(* IEC 61131-3 sources: Mizera_Tube/Plc (part 15) *)

(* ---- StatMReg.plc ---- *)
#funcdec "DynMng.plc"

VAR
JUMP_INT:       LINEAR_CALC;
END_VAR

VAR_IN_OUT
PercentOutRng  AT %LSRCostK17;
END_VAR

FUNCTION_BLOCK REG_STATE_MACHINE

VAR
command:                DWORD;
State:                  DWORD;
LastCutDistance:        DWORD;
SetPointOutRange:       DWORD;      * PLC monitoring about set point out of range
RegFrozen:               BOOL;      * Regulation has been frozen from post processor
autoRegJump:             BOOL;
JumpinMode:              BOOL;
JumpinL3Mode:            BOOL;

autoRegL10:              BOOL;
L10Mode:                 BOOL;

QJump:                  DWORD;
VettYTot:               DWORD;
VettXTot:               DWORD;
VettCTot:               DWORD;

DistTot:                DWORD;
ActualDistTot:          DWORD;
ActualYDist:            DWORD;
ActualXDist:            DWORD;
ActualCDist:            DWORD;
DeltaSetPoint:          DWORD;
ZLinInterp:             DWORD;

TON_TIME_OUT:             TON;
TON_ProbeTo:              TON;
APPOGGIO:               DWORD;
appoggio:               DWORD;

firScan:                DWORD;
firScan1:               DWORD;
delScan:                DWORD;
error1:                 DWORD;
error2:                 DWORD;
error3:                 DWORD;
ToolFlt_Q_FILTERED:     DWORD;
ToolFlt_Q_FILTERED1:    DWORD;
ToolFlt_Q_FILTERED_DEL: DWORD;
ThrForOutRange:         DWORD;
SetP_S_BeforeHold:      DWORD;
tem_PercentOutRng:      DWORD;

ActualXDist_A:          DWORD;
ActualYDist_A:          DWORD;
ActualZDist_A:          DWORD;
ActualCDist_A:          DWORD;
Actual_Dist_A:          DWORD;
ActualXDist_B:          DWORD;
ActualYDist_B:          DWORD;
ActualZDist_B:          DWORD;
ActualCDist_B:          DWORD;
Actual_Dist_B:          DWORD;
Par:                   DWORD;

END_VAR

VAR_INPUT

xFirstPlcHandling:       BOOL;
xStartEx:                BOOL;
xFreezeRegol:            BOOL;         * External command to freeze regulation
xMove_Z:                   BOOL;
xHold:                   BOOL;
xFirstFirCost:          DWORD;         * ms
xSecondFirCost:         DWORD;         * ms
xDelayCost:             DWORD;         * ms
xMove_Z_SetP:             DWORD;

xProbThres:             DWORD;
xZ_TCP:                 DWORD;
xSetpoint:              DWORD;
xIsoPhase:              DWORD;         * 1: probing phase, 2: Piercing ,4: Cutting
xSensorRange:           DWORD;         * Max ange of the sensor

xNextPos_X_Jump:        DWORD;         * X setpoint coordinate for jump
xNextPos_Y_Jump:        DWORD;         * Y setpoint coordinate for jump
xNextPos_C_Jump:        DWORD;         * C setpoint coordinate for jump
xNextPos_Z_Jump:        DWORD;         * C setpoint coordinate for jump
xInit_X_Posit:          DWORD;         * X init jump position
xInit_Y_Posit:          DWORD;         * Y init jump position
xInit_C_Posit:          DWORD;         * C init jump position
xInit_Z_Posit:          DWORD;         * Z init jump position
xActual_X_Posit:        DWORD;         * X Actual position
xActual_Y_Posit:        DWORD;         * Y Actual position
xActual_C_Posit:        DWORD;         * C Actual position
xActual_Z_Posit:        DWORD;         * Z Actual position
xNextSetp:              DWORD;         * Setpoint after jump
xPrevSetp:              DWORD;         * setpoint before jump
xDistEnabRegul:         DWORD;         * Distance from target to enab regulation during jump
xZDistStopProbeJ:       DWORD;         * Z dstance to disable Probe mode during jump
xJumpReq:               BOOL;          * Jump request from ISO
xJumpL3Req:             BOOL;          * Jump L3 request from ISO
xL10Req:                BOOL;          * L10 Request from ISO
xCosBevelAngle:         DWORD;

* Surface VRTC
xSurfSignalLock:         BOOL;
xSurfaceBusy:            BOOL;
xISO_S_SimEnab:          BOOL;
xISO_S_ErrAmp:           BOOL;

* Tool VRTC

xToolSignalLock:         BOOL;
xToolBusy:               BOOL;
xISO_T_SimEnab:          BOOL;
xISO_T_ErrAmp:           BOOL;
xISO_T_SetPoint:        DWORD;
xToolFlt_Q:             DWORD;
END_VAR

VAR_OUTPUT
* Surface_VRTC_Out
y_S_SimEnab:            BOOL;             * Put Surface vrtc in Simulation
y_S_ErrAmp:             BOOL;             * Surface Error Amplifier
y_S_SetPoint:          DWORD;             * surface setpoint

* Tool_VRTC_Out
y_T_SimEnab:            BOOL;             * disable T vrtc simulation
y_T_ErrAmp:             BOOL;             * Tool Error Amplifier
y_T_SetPoint:          DWORD;

* General
yComRunning:            BOOL;
yWait:                  BOOL;
yIncSetPReached:        BOOL;
yL3SetpointReached:     BOOL;

yVPBSelect:            DWORD;
yStateMachinePhase:    DWORD;
yState:                DWORD;

END_VAR

* Reset variables at the first plc handling command

LD   xFirstPlcHandling
JMPCN no_default

LD   xFirstFirCost
DIV  %plc0.PlcCycle         * plc scan
ST   firScan

LD   xSecondFirCost
DIV  %plc0.PlcCycle         * plc scan
ST   firScan1                      **

LD   xDelayCost
DIV  %plc0.PlcCycle         * plc scan
ST   delScan                      **

LD   0
FIR_INIT (INS=1, LEN=firScan)
ST   error1

LD   0
FIR_INIT (INS=2, LEN=firScan1)
ST   error2

LD   0
DELAY_INIT (INS=1, LEN=delScan)
ST   error3
*

LD   xISO_S_SimEnab
ST   y_S_SimEnab

LD   xISO_S_ErrAmp
ST   y_S_ErrAmp

LD   xISO_T_SimEnab
ST   y_T_SimEnab

LD   xISO_T_ErrAmp
ST   y_T_ErrAmp

LD   xISO_T_SetPoint
ST   y_T_SetPoint
ST   LastCutDistance

LD   0
ST   State
ST   y_S_SetPoint                 * surface setpoint
ST   yVPBSelect
ST   yComRunning
ST   xStartEx
ST   yStateMachinePhase
ST   xJumpReq
ST   RegFrozen
ST   QJump
ST   %M180
ST   JumpinMode
ST   JumpinL3Mode
ST   yWait
ST   yIncSetPReached
ST   %PLCmsg0.8
no_default:

* Machine filters and delay model ALWAYS REFRESHED

LD   0                       * N/C
FIR_RUN (INS=1, X=xToolFlt_Q)
ST      ToolFlt_Q_FILTERED1

LD   0                       * N/C
FIR_RUN (INS=2, X=ToolFlt_Q_FILTERED1)
ST      ToolFlt_Q_FILTERED

LD   0
DELAY_RUN (INS=1,X=ToolFlt_Q_FILTERED)
DIV  10
ST  ToolFlt_Q_FILTERED_DEL

*

* Cut Distance Out of range monitoring

LD   PercentOutRng
ST   tem_PercentOutRng

LD   PercentOutRng
GT   70
OR(
LD   PercentOutRng
LT   15
)
JMPCN _SAFERNG
     LD   70
     ST   tem_PercentOutRng
_SAFERNG:

LD   xSensorRange
MULDIV (M=tem_PercentOutRng,D=1000)           * 70% del range del sensore
ST   ThrForOutRange

LD   xSetpoint
GT   ThrForOutRange
ST   SetPointOutRange

*-----------------------------------------------------------------------------------------
* Probing state machine

LD   State
EQ   0
JMPCN STATE0_end
STATE0:

 * Operative mode change

 LD    xIsoPhase
 EQ    2
 ANDN  JumpinMode
 ANDN  JumpinL3Mode
 JMPCN no_piercing_state
  LD   200                 * Piercing in progress
  ST   State
  JMP state_machine_end
 no_piercing_state:

 LD    xIsoPhase
 EQ    4
 ANDN  JumpinMode
 ANDN  JumpinL3Mode
 JMPCN no_cut_state
  LD   300                 * Cutting in progress
  ST   State
  JMP state_machine_end
 no_cut_state:

 LD    xHold
 JMPCN no_hold_sim
  LD   20                 * Go in hold condition and stop the VRTC
  ST   State
  JMP state_machine_end
 no_hold_sim:

 *
 LD    xIsoPhase
 ST    yStateMachinePhase

 *
 */////////////////////////////////////////////////////////////////////////////////
 *// Probing: vrtc wait the Z axis position threshold and disable the surface
 *// vrtc simulation and put the correct setpoint
 */////////////////////////////////////////////////////////////////////////////////

 LD    xIsoPhase
 EQ    1                                   *
 ANDN  (
 LD    xZ_TCP
 LT    xProbThres
 OR    %C18.17                             * Capacitive test in progress
 )
 AND   xStartEx
 ST    appoggio
 CAL   TON_ProbeTo(IN=appoggio,PT=10000)   * 10s
 LD    TON_ProbeTo.Q
 S     %PLCmsg0.8

 LD    xIsoPhase
 EQ    1                                   *
 AND   (
 LD    xZ_TCP
 LT    xProbThres
 OR    %C18.17                             * Capacitive test in progress
 )
 AND   xStartEx
 JMPCN STATE0_endif_A

  LD   1
  R    y_S_SimEnab                         * Put Surface vrtc in Simulation

  LD   2
  ST   yVPBSelect

  LD   xToolFlt_Q
  DIV  10
  MULDIV(M=xCosBevelAngle,D=1000)
  ST   y_S_SetPoint                        * surface setpoint

  LD   1
  ST   yComRunning

  LD  10
  ST  State
  JMP state_machine_end
 STATE0_endif_A:
*///////////////////////////////////////////////////////////////////////////////
JMP state_machine_end
STATE0_end:

LD   State
EQ   10
JMPCN STATE10_end
STATE10:
*/////////////////////////////////////////////////////////////////////////////////
*// Wait the position is reached from surface vrtc
*/////////////////////////////////////////////////////////////////////////////////

 LD    xHold
 JMPCN no_hold_real
  LD   30                 * Go in hold condition and stop the VRTC
  ST   State
  JMP state_machine_end
 no_hold_real:

 LD   xSurfSignalLock
 ANDN xSurfaceBusy
 ANDN xStartEx
 JMPCN STATE10_endif_A

  LD   0
  ST   yComRunning

  LD   0
  ST   State
  JMP state_machine_end
 STATE10_endif_A:
*///////////////////////////////////////////////////////////////////////////////
JMP state_machine_end
STATE10_end:

* During hold not allow VRTC movement

LD   State
EQ   20
JMPCN STATE20_end
STATE20:
*/////////////////////////////////////////////////////////////////////////////////
*// Hold the Z axis during the simulated descendent trajectory
*/////////////////////////////////////////////////////////////////////////////////

 LD   1
 R    y_S_ErrAmp

 LDN   xHold
 JMPCN STATE20_endif_A

  LD   1
  S    y_S_ErrAmp

  LD   0
  ST   State

  JMP state_machine_end
 STATE20_endif_A:

*///////////////////////////////////////////////////////////////////////////////
JMP state_machine_end
STATE20_end:

*
LD   State
EQ   30
JMPCN STATE30_end
STATE30:
*/////////////////////////////////////////////////////////////////////////////////
*// Hold the Z axis during the real descendent trajectory
*/////////////////////////////////////////////////////////////////////////////////

 LD   1
 R    y_S_ErrAmp

 LDN   xHold
 JMPCN STATE30_endif_A

  LD   1
  S    y_S_ErrAmp

  LD   10
  ST   State

  JMP state_machine_end
 STATE30_endif_A:

*///////////////////////////////////////////////////////////////////////////////
JMP state_machine_end
STATE30_end:

*-----------------------------------------------------------------------------------------

*-----------------------------------------------------------------------------------------
* Piercing state

LD   State
EQ   200
JMPCN STATE200_end
STATE200:
*/////////////////////////////////////////////////////////////////////////////////
*// Set piercing vpb selector
*/////////////////////////////////////////////////////////////////////////////////

 LD   xIsoPhase
 EQ   2
 ANDN xToolBusy            * update
 ANDN xSurfaceBusy         * update
 JMPCN STATE200_endif_A

  LD   3
  ST   yVPBSelect

  LD   1
 * R    y_T_SimEnab                         * Enable Tool Vrtc simulation
  S    y_T_SimEnab                         * Enable Tool Vrtc simulation

  LD   1
* S    y_S_SimEnab                         * Enable Surface vrtc Simulation
  R    y_S_SimEnab                         * Enable Surface vrtc Simulation

  LD  210
  ST  State
  JMP state_machine_end
 STATE200_endif_A:
*///////////////////////////////////////////////////////////////////////////////
JMP state_machine_end
STATE200_end:

LD   State
EQ   210
JMPCN STATE210_end
STATE210:

 * Operative mode change

 LD    xIsoPhase
 EQ    4
 JMPCN no_cut_state1
  LD    300                 * Cutting in progress
  ST    State
  JMP state_machine_end
 no_cut_state1:
*/////////////////////////////////////////////////////////////////////////////////
*// Change setpoint during piercing and synchronize the Piercing state with
*// Iso.
*/////////////////////////////////////////////////////////////////////////////////

 LD   xIsoPhase
 ST   yStateMachinePhase

 LD   xIsoPhase
 EQ   2
 AND  xStartEx
 ANDN xToolBusy
 ANDN xSurfaceBusy
 JMPCN STATE210_endif_A

  ** TEST  : in case there is a switch from out of range to in range
   LD   3
   ST   yVPBSelect
  **
  LD   1
** R    y_T_SimEnab                        * Enable Tool Vrtc simulation
  S    y_T_SimEnab                        * Enable Tool Vrtc simulation

  LD   1
** S    y_S_SimEnab                         * Enable Surface vrtc Simulation
  R    y_S_SimEnab                         * Enable Surface vrtc Simulation

  LD  SetPointOutRange                    *
  JMPCN no_sim_tool
  ** TEST
   LD   6
   ST   yVPBSelect
  **

   LD   1
   S    y_T_SimEnab                       * Enable Tool Vrtc simulation

   LD   1
*  S    y_S_SimEnab                         * Enable Surface vrtc Simulation
   S    y_S_SimEnab                         * Enable Surface vrtc Simulation

  no_sim_tool:

  LD  xSetpoint
  ST  y_T_SetPoint                        * Tool setpoint
  ST  LastCutDistance

  LD  1
  ST  yComRunning

  LD  220
  ST  State
  JMP state_machine_end
 STATE210_endif_A:
*///////////////////////////////////////////////////////////////////////////////
JMP state_machine_end
STATE210_end:

LD   State
EQ   220
JMPCN STATE220_end
STATE220:
*/////////////////////////////////////////////////////////////////////////////////
*// Setpoint reached:end of the command is set and fo to state 210 ready for
*// for next change
*/////////////////////////////////////////////////////////////////////////////////

 LD   ToolFlt_Q_FILTERED_DEL
 LT   ThrForOutRange
 AND (
  LD  LastCutDistance
  LT  ThrForOutRange
  )
 JMPCN no_setp_copy5

  LD   3
  ST   yVPBSelect

  LD   1
  R    y_S_SimEnab                         * Put Surface vrtc in Simulation

  LD   ToolFlt_Q_FILTERED_DEL
  MULDIV(M=xCosBevelAngle,D=1000)
  ST   y_S_SetPoint                       * Surface setpoint

 no_setp_copy5:

** LD   xToolSignalLock
** ANDN xToolBusy
 LD   xSurfSignalLock
 ANDN xSurfaceBusy
 ANDN xStartEx
 JMPCN STATE220_endif_A

**  LD  xSetpoint
**  ST  LastCutDistance

  LD  0
  ST  yComRunning

 ** LD   1
 ** S    y_T_SimEnab                       * Enable Tool Vrtc simulation

  LD  210
  ST  State
  JMP state_machine_end
 STATE220_endif_A:
*///////////////////////////////////////////////////////////////////////////////
JMP state_machine_end
STATE220_end:

*-----------------------------------------------------------------------------------------
* Cutting phase

LD   State
EQ   300
JMPCN STATE300_end
STATE300:

 LD  xIsoPhase
 ST  yStateMachinePhase
*/////////////////////////////////////////////////////////////////////////////////
*// This is a transition state in order to set the surface vrtc ready for
*// regulation. If the setpoint is out of range S vrtc will be in simulation.
*//
*/////////////////////////////////////////////////////////////////////////////////
 LD  xIsoPhase
 EQ  4
 ANDN xToolBusy            * update
 ANDN xSurfaceBusy         * update
 JMPCN STATE300_endif_A

  LD   1
  S    y_T_SimEnab                        * Enable Tool Vrtc simulation

  LD   1
  R    y_S_SimEnab                        * Put Surface vrtc in Simulation

  LD   4
  ST   yVPBSelect

  LD   310
  ST   State

  LD  SetPointOutRange
  JMPCN no_sim_surf
   LD   1
   S    y_S_SimEnab                       * Put Surface vrtc in Simulation
   JMP state_machine_end
  no_sim_surf:
* If the surface vrtc is in simulation not change the setpoint, otherwise it will wrong the surface position

  LD   ToolFlt_Q_FILTERED_DEL
  MULDIV(M=xCosBevelAngle,D=1000)
  ST   y_S_SetPoint                       * Surface setpoint

  JMP state_machine_end
 STATE300_endif_A:
*///////////////////////////////////////////////////////////////////////////////
JMP state_machine_end
STATE300_end:

LD   State
EQ   310
JMPCN STATE310_end
STATE310:
*/////////////////////////////////////////////////////////////////////////////////
*// Cutting mode idle: from this state is possible freeze and unfreeze regulation,
*// manage runtime setpoint change and jump request
*/////////////////////////////////////////////////////////////////////////////////

 LD   ToolFlt_Q_FILTERED_DEL
 LT   ThrForOutRange
 AND (
  LD  LastCutDistance
  LT  ThrForOutRange
  )
 ANDN RegFrozen
 ANDN L10Mode
 ANDN JumpinMode
 ANDN JumpinL3Mode
 JMPCN no_setp_copy

  LD   4
  ST   yVPBSelect

  LD   1
  R    y_S_SimEnab                         * Put Surface vrtc in Simulation

  LD   ToolFlt_Q_FILTERED_DEL
  MULDIV(M=xCosBevelAngle,D=1000)
  ST   y_S_SetPoint                       * Surface setpoint

 no_setp_copy:

* Reset L5 Routine

 LDN  xJumpReq
 JMPCN no_res_jump
  LD  1
  R   JumpinMode
 no_res_jump:

 * Reset L3 Routine

 LDN  xJumpL3Req
 JMPCN no_res_jumpL3
  LD  1
  R   JumpinL3Mode
 no_res_jumpL3:

* Reset L10 Routine

 LDN  xL10Req
 JMPCN no_res_L10
  LD  1
  R   L10Mode
 no_res_L10:

* Change operative mode to Piercing

 LD    xIsoPhase
 EQ    2
 ANDN  JumpinMode
 ANDN  JumpinL3Mode
 ANDN  L10Mode
 JMPCN no_piercing_state1
  LD   200                 * Piercing in progress
  ST   State
  JMP state_machine_end
 no_piercing_state1:

* Managment of freeze regulation from post processor
* Freeze Regulation
 LD   xFreezeRegol
 ANDN RegFrozen
 JMPCN no_freeze_en
  LD  330
  ST  State
  JMP state_machine_end *
 no_freeze_en:

* Jumping Request

 LD   xJumpReq
 ANDN JumpinMode
 ANDN JumpinL3Mode
 ANDN L10Mode
 JMPCN no_jump_req

  LD  1
  S   JumpinMode

  LD  350
  ST  State
  JMP state_machine_end
 no_jump_req:
*

* Jumping L3 Request

 LD   xJumpL3Req
 ANDN JumpinMode
 ANDN L10Mode
 JMPCN no_jump_reqL3

  LD  1
  S   JumpinL3Mode

  LD  430
  ST  State
  JMP state_machine_end
 no_jump_reqL3:
*

* L10 Request (used for cutting to piercing height)

 LD   xL10Req
 ANDN JumpinMode
 ANDN JumpinL3Mode
 ANDN L10Mode
 JMPCN no_L10_req

  LD  1
  S   L10Mode

  LD  370
  ST  State
  JMP state_machine_end
 no_L10_req:
*
* Hold Request During cut

 LD   xMove_Z
 JMPCN no_hold_req

  LD  y_S_SetPoint
  ST  SetP_S_BeforeHold

  LD  400
  ST  State
  JMP state_machine_end
 no_hold_req:

*
*/////////////////////////////////////////////////////////////////////////////////
*// If the cut distance need to be changed, this state
*// enable the simulation on the surface vrtc, disable simulation on tool vrtc
*// and set the new setpoint
*/////////////////////////////////////////////////////////////////////////////////

 LD   LastCutDistance
 NE   xSetpoint
 JMPCN STATE310_endif_A

  LD   1
  R    y_S_SimEnab                         * Put Surface vrtc in Simulation

  LD   1
  S    y_T_SimEnab                         * Enable Tool Vrtc simulation

  LD   xSetpoint
  ST   y_T_SetPoint                        * Tool setpoint
  ST   LastCutDistance                     * new

  LD   320
  ST   State

  LD  ToolFlt_Q_FILTERED_DEL
  GT  ThrForOutRange                    *
  OR  RegFrozen
  OR (
  LD  xSetpoint
  GT  ThrForOutRange
  )
  JMPCN no_sim_tool1
   ** TEST :set simulated vrtc parameters
   LD   6
   ST   yVPBSelect
   **

   LD   1
   S    y_S_SimEnab                        * Put Surface vrtc in Simulation
  JMP state_machine_end
  no_sim_tool1:

  LD   ToolFlt_Q_FILTERED_DEL
  MULDIV(M=xCosBevelAngle,D=1000)
  ST   y_S_SetPoint                       * Surface setpoint

  JMP state_machine_end
 STATE310_endif_A:

* Enable regulation Request
* This request must be here in order to not exchange the order of
* the command with the set point change

 LDN  xFreezeRegol
 AND  RegFrozen
 JMPCN no_freeze_dis
  LD  340
  ST  State
  JMP state_machine_end
 no_freeze_dis:

*///////////////////////////////////////////////////////////////////////////////
JMP state_machine_end
STATE310_end:

LD   State
EQ   320
JMPCN STATE320_end
STATE320:
*/////////////////////////////////////////////////////////////////////////////////
*// Wait the position is reached RUN-TIME. Added a  time-out condition
*/ to avoid the regulation stack on the reaching of one setpoint
*/////////////////////////////////////////////////////////////////////////////////

  LD   ToolFlt_Q_FILTERED_DEL
  LT   ThrForOutRange
  AND (
   LD  LastCutDistance
   LT  ThrForOutRange
   )
  ANDN RegFrozen
  JMPCN no_setp_copy1
   ** TEST
   LD   4
   ST   yVPBSelect
   **

   LD   1
   R    y_S_SimEnab                         * Put Surface vrtc in Simulation

   LD   ToolFlt_Q_FILTERED_DEL
   MULDIV(M=xCosBevelAngle,D=1000)
   ST   y_S_SetPoint                       * Surface setpoint
  no_setp_copy1:

  LDN  xToolSignalLock
  ANDN xToolBusy
  ST   appoggio

* Time-out is mandatory, in order to avoid the regulation keep this state
* and saturate the vrtc limit

  CAL  TON_TIME_OUT (IN:=appoggio,PT:=250)

  LD   xToolSignalLock
  ANDN xToolBusy
  OR   TON_TIME_OUT.Q
  JMPCN STATE320_endif_A
    ** TEST
    LD   4
    ST   yVPBSelect
    **

    LD   1
    R    y_S_SimEnab                         * Put Surface vrtc in Simulation

    LD   1
    S    y_T_SimEnab                         * Enable Tool Vrtc simulation

    LD   310
    ST   State

    LD  SetPointOutRange               **** Verificare se va aggiornato con le condizioni fatte per gli altri stati
    OR  RegFrozen
    JMPCN no_sim_surf1
     ** TEST
     LD   6
     ST   yVPBSelect
     **

     LD   1
     S    y_S_SimEnab                       * Put Surface vrtc in Simulation
     JMP state_machine_end
    no_sim_surf1:

* If the surface vrtc is in simulation not change the setpoint, otherwise it will wrong the surface position

   LD   ToolFlt_Q_FILTERED_DEL
   MULDIV(M=xCosBevelAngle,D=1000)
   ST   y_S_SetPoint                       * Surface setpoint

 JMP state_machine_end
 STATE320_endif_A:
*///////////////////////////////////////////////////////////////////////////////
JMP state_machine_end
STATE320_end:

LD   State
EQ   330
JMPCN STATE330_end
STATE330:
*/////////////////////////////////////////////////////////////////////////////////
*// Enable the simulation of the sensor when post processor need freeze
*// the height control
*/////////////////////////////////////////////////////////////////////////////////

 ** TEST
 LD   6
 ST   yVPBSelect
 **

 LD  1
 S   y_S_SimEnab                       * Put Surface vrtc in Simulation

 LD  1
 S   y_T_SimEnab                         * Enable Tool Vrtc simulation

 LD  1
 S   RegFrozen

 LD  310
 ST  State

 JMP state_machine_end
STATE330_endif_A:
*///////////////////////////////////////////////////////////////////////////////
JMP state_machine_end
STATE330_end:

LD   State
EQ   340
JMPCN STATE340_end
STATE340:
*/////////////////////////////////////////////////////////////////////////////////
*// Post processor command regulation again, but need to be careful about set point
*// if it is inside the range, surface can back to regulate otherwise no
*/////////////////////////////////////////////////////////////////////////////////

  LD   ToolFlt_Q_FILTERED_DEL
  LT   ThrForOutRange
  AND (
   LD  LastCutDistance
   LT  ThrForOutRange
   )
 JMPCN no_remove_sim_S
  ** TEST
  LD   4
  ST   yVPBSelect
  **

  LD  1
  R   y_S_SimEnab                        * Surface vrtc in Simulation

* Need give setpoint because if it change distance when is frozen and setpoint is inside the range
* it is not refresced on surface regulator

  LD   ToolFlt_Q_FILTERED_DEL
  MULDIV(M=xCosBevelAngle,D=1000)
  ST   y_S_SetPoint                      * Surface setpoint

 no_remove_sim_S:

 LD  1
 S   y_T_SimEnab                         * Enable Tool Vrtc simulation

 LD  1
 R   RegFrozen

 LD  310
 ST  State

 JMP state_machine_end
STATE340_endif_A:
*///////////////////////////////////////////////////////////////////////////////
JMP state_machine_end
STATE340_end:

* Jump
LD   State
EQ   350
JMPCN STATE350_end
STATE350:
*/////////////////////////////////////////////////////////////////////////////////
*// Jump Request: select VPBselect at 1 for jump column,put vrtc surface in
*// simulation. The algorithm calulates the setpoint for Surface and Tool
*// Vrtc. Surface will perform the parabolic trajectory, the Tool will apply the
*// setpoint change
*/////////////////////////////////////////////////////////////////////////////////
 LD  xStartEx
 JMPCN no_start_jump

  LD   1
  ST   yComRunning

  LD   1
  ST   yVPBSelect

  LD   1
  S    y_S_SimEnab              * Surface vrtc in Simulation

  LD   xNextPos_Y_Jump         * Y setpoint coordinate for jump
  SUB  xInit_Y_Posit           * Y init jump position
  ABS
  ST   VettYTot                * Distance in Y direction

  LD   xNextPos_X_Jump         * X setpoint coordinate for jump
  SUB  xInit_X_Posit           * X init jump position
  ABS
  ST   VettXTot                * Distance in X direction

  LD   0
  ST   VettCTot                      ** Distance in C direction

  LD   xNextPos_C_Jump
  SUB  xInit_C_Posit
  ABS
  ST   VettCTot                      ** Distance in C direction

  LD   0
  HYPOT (X=VettXTot,Y=VettYTot)
  ST   DistTot                 * total distance for jump

  LD   0
  HYPOT (X=DistTot,Y=VettCTot)       ** total distance for jump
  ST   DistTot                       ** total distance for jump

  LD   xActual_X_Posit
  SUB  xInit_X_Posit                 * X init jump position
  ABS
  ST   ActualXDist

  LD   xActual_Y_Posit               * Y Actual position
  SUB  xInit_Y_Posit                 * Y init jump position
  ABS
  ST   ActualYDist

  LD   xActual_C_Posit
  SUB  xInit_C_Posit
  ABS
  ST   ActualCDist

  LD   0
  HYPOT (X=ActualXDist,Y=ActualYDist)
  ST   ActualDistTot

  LD   0
  HYPOT (X=ActualDistTot,Y=ActualCDist)
  ST   ActualDistTot
  ST   %M181

  * Calcolo quota per jumping mode

  LD   ActualDistTot
  ST   JUMP_INT.xInput               * Distance to go

  LD   130
  ST   JUMP_INT.xIndex               * cut line index (initial value 1 to 10)

  CAL  JUMP_INT

  LD   JUMP_INT.yResult              * Result
  DIV  10
  ST   QJump                         ** Quota Z per Jumping

  LD   xPrevSetp                      * setpoint before jump
  DIV  10
  ADD  QJump
  ST   y_S_SetPoint
  ST   %M184

  ************************************************************************************
*  Algorithm for auto jump regulation enable
*  and setpoint changing compensation

  LD   xNextSetp                * Setpoint after jump
  SUB  xPrevSetp                * setpoint before jump
  ST   DeltaSetPoint

* TEST
 * LD   ActualDistTot
 * MUL  2
 * ST   APPOGGIO

 * LD   APPOGGIO
 * GT   DistTot
 * JMPCN forcedist
 *  LD   DistTot
 *  ST   APPOGGIO
 * forcedist:
***
 * LD   APPOGGIO
  LD   ActualDistTot
  MULDIV (M=DeltaSetPoint,D=DistTot) ** total distance for jump
  DIV  10                            *cmm
  ST   ZLinInterp

  LD   xPrevSetp                * setpoint before jump
  DIV  10
  ADD  ZLinInterp
  ST   y_T_SetPoint

  ** Test of regulation on fly

  LD   DistTot                       ** total distance for jump
  SUB  ActualDistTot                 * Actual total distance by measured speed
  LE   xDistEnabRegul                * Distance from target to enab regulation
  ST   autoRegJump                   ** During jump allow auto regulation on

  LD   autoRegJump
  JMPCN no_jump_end

    LD  xZ_TCP
    GT  xZDistStopProbeJ             * distance along Z to disable the probe vpbselector during jump
    JMPCN no_Zover_range

     LD  0
     ST  yVPBSelect

     LD   xPrevSetp                * setpoint before jump
     DIV  10
     MULDIV(M=xCosBevelAngle,D=1000)
     ST  y_S_SetPoint

    JMP no_jump_end
    no_Zover_range:

    LD  1
    R   y_S_SimEnab                 * Surface vrtc in Simulation

    LD  2
    ST  yVPBSelect

    LD   ToolFlt_Q_FILTERED_DEL
    MULDIV(M=xCosBevelAngle,D=1000)
    ST  y_S_SetPoint
    ST  %M183

  no_jump_end:
 no_start_jump:

 LDN  xJumpReq
 JMPCN no_end_jump

  LD  1
  R   y_S_SimEnab                 * Surface vrtc in Simulation

  LD  2
  ST  yVPBSelect

  LD   ToolFlt_Q_FILTERED_DEL
  MULDIV(M=xCosBevelAngle,D=1000)
  ST  y_S_SetPoint

  LD  360
  ST  State
 no_end_jump:

 JMP state_machine_end
STATE350_endif_A:
*///////////////////////////////////////////////////////////////////////////////
JMP state_machine_end
STATE350_end:

LD   State
EQ   360
JMPCN STATE360_end
STATE360:
*/////////////////////////////////////////////////////////////////////////////////
*// Wait the position is reached after jump
*/////////////////////////////////////////////////////////////////////////////////

 LD   ToolFlt_Q_FILTERED_DEL
 MULDIV(M=xCosBevelAngle,D=1000)
 ST  y_S_SetPoint

 LD   xSurfSignalLock
 ANDN xSurfaceBusy
 ANDN xStartEx
 JMPCN STATE360_endif_A

    LD   0
    ST   yComRunning

    LD   xNextSetp                * Setpoint after jump
    DIV  10
    ST   LastCutDistance

    LD   1                        * Reset bit to enable always regulation after jump
    R    RegFrozen

    LD   310
    ST   State
 JMP state_machine_end
STATE360_endif_A:
*///////////////////////////////////////////////////////////////////////////////
JMP state_machine_end
STATE360_end:

LD   State
EQ   370
JMPCN STATE370_end
STATE370:
*/////////////////////////////////////////////////////////////////////////////////
*// This state manage the L10 cutting transition, to reach the set point it is only
*// interpolated the Tool VRTC from cutting position to Piercing position.
*/////////////////////////////////////////////////////////////////////////////////

 LD  xStartEx
 JMPCN no_start_L10

  LD   1
  ST   yComRunning

  LD   1
  ST   yVPBSelect

  LD   1
  S    y_S_SimEnab              * Surface vrtc in Simulation

  LD   xNextPos_Y_Jump         * Y setpoint coordinate for jump
  SUB  xInit_Y_Posit           * Y init jump position
  ABS
  ST   VettYTot                * Distance in Y direction

  LD   xNextPos_X_Jump         * X setpoint coordinate for jump
  SUB  xInit_X_Posit           * X init jump position
  ABS
  ST   VettXTot                * Distance in X direction

  LD   0
  HYPOT (X=VettXTot,Y=VettYTot)
  ST   DistTot                 * total distance for jump

  LD   xActual_X_Posit
  SUB  xInit_X_Posit                 * X init jump position
  ABS
  ST   ActualXDist

  LD   xActual_Y_Posit               * Y Actual position
  SUB  xInit_Y_Posit                 * Y init jump position
  ABS
  ST   ActualYDist

  LD   0
  HYPOT (X=ActualXDist,Y=ActualYDist)
  ST   ActualDistTot
  ST   %M181

  ************************************************************************************
*  Algorithm for auto jump regulation enable
*  and setpoint changing compensation

  LD   xNextSetp                * Setpoint after jump
  SUB  xPrevSetp                * setpoint before jump
  ST   DeltaSetPoint

* TEST
 * LD   ActualDistTot
 * MUL  2
 * ST   APPOGGIO

 * LD   APPOGGIO
 * GT   DistTot
 * JMPCN forcedist1
 *  LD   DistTot
 *  ST   APPOGGIO
 * forcedist1:
***
  *LD   APPOGGIO
  LD   ActualDistTot
  MULDIV (M=DeltaSetPoint,D=DistTot) ** total distance for jump
  DIV  10                            *cmm
  ST   ZLinInterp

  LD   xPrevSetp                * setpoint before jump
  DIV  10
  ADD  ZLinInterp
  ST   y_T_SetPoint

  ** Test of regulation on fly

  LD   DistTot                       ** total distance for jump
  SUB  ActualDistTot                 * Actual total distance by measured speed
  LE   xDistEnabRegul                * Distance from target to enab regulation
  ST   autoRegL10                   ** During jump allow auto regulation on

  LD   autoRegL10
  JMPCN no_L10_end

    LD  1
    R   y_S_SimEnab                 * Surface vrtc in Simulation

    LD  2
    ST  yVPBSelect

    LD   ToolFlt_Q_FILTERED_DEL
    MULDIV(M=xCosBevelAngle,D=1000)
    ST  y_S_SetPoint
    ST  %M183

  no_L10_end:
 no_start_L10:

 LDN  xL10Req
 JMPCN no_end_L10

  LD  1
  R   y_S_SimEnab                 * Surface vrtc in Simulation

  LD  2
  ST  yVPBSelect

  LD   ToolFlt_Q_FILTERED_DEL
  MULDIV(M=xCosBevelAngle,D=1000)
  ST  y_S_SetPoint

  LD  380
  ST  State
 no_end_L10:

 JMP state_machine_end
STATE370_endif_A:
*///////////////////////////////////////////////////////////////////////////////
JMP state_machine_end
STATE370_end:
*
LD   State
EQ   380
JMPCN STATE380_end
STATE380:
*/////////////////////////////////////////////////////////////////////////////////
*// Wait the position is reached after L10
*/////////////////////////////////////////////////////////////////////////////////

 LD   ToolFlt_Q_FILTERED_DEL
 MULDIV(M=xCosBevelAngle,D=1000)
 ST  y_S_SetPoint

 LD   xSurfSignalLock
 ANDN xSurfaceBusy
 ANDN xStartEx
 JMPCN STATE380_endif_A

    LD   0
    ST   yComRunning

    LD   xNextSetp                * Setpoint after jump       CAMBIARE NOME
    DIV  10
    ST   LastCutDistance

    LD   310
    ST   State
 JMP state_machine_end
STATE380_endif_A:
*///////////////////////////////////////////////////////////////////////////////
JMP state_machine_end
STATE380_end:

* Hold

LD   State
EQ   400
JMPCN STATE400_end
STATE400:
*///////////////////////////////////////////////////////////////////////////////////
*// Hold management: Z is moved according the Z inc movement; when xZmove is
*// removed, the Z back in the prevous point. If the operator move by retrace
*// the tool setpoint is updated run-time, the freeze conditition due to the
*// M82 M83 or distance out of range that can happen during the retrace are managed.
*///////////////////////////////////////////////////////////////////////////////////

  LD  1
  S   y_S_SimEnab                 * Surface vrtc in Simulation

  LD  xMove_Z_SetP
  ST  y_S_SetPoint

  LD  5
  ST  yVPBSelect

  LD  xSetpoint
  ST  y_T_SetPoint
  ST  LastCutDistance

  LD  xFreezeRegol
  ST  RegFrozen

  LDN  yIncSetPReached
  JMPCN no_wait_incSetp
    LD   410
    ST   State
    JMP  state_machine_end
  no_wait_incSetp:

  LDN  xMove_Z
  JMPCN no_return_pause

    LD  1
    S   yWait

* IF stand-off is in capacitive range

    LD  ToolFlt_Q_FILTERED_DEL
    LT  ThrForOutRange
    AND (
    LD  LastCutDistance
    LT  ThrForOutRange
    )
    ANDN RegFrozen
    JMPCN no_setp_copy3
    ** TEST
     LD   5
     ST   yVPBSelect
    **
     LD   1
     R    y_S_SimEnab                        * Put Surface vrtc in Simulation

     LD   ToolFlt_Q_FILTERED_DEL
     MULDIV(M=xCosBevelAngle,D=1000)
     ST   y_S_SetPoint                       * Surface setpoint

     LD   420
     ST   State
    JMP state_machine_end
    no_setp_copy3:

    LD  ToolFlt_Q_FILTERED_DEL
    GT  ThrForOutRange
    OR (
    LD  LastCutDistance
    GT  ThrForOutRange
    )
    OR  RegFrozen
    JMPCN no_setp_copy4

     **
     LD   5
     ST   yVPBSelect
     **
     LD   1
     S    y_S_SimEnab                        * Put Surface vrtc in Simulation

     LD   SetP_S_BeforeHold
     ST   y_S_SetPoint                       * Surface setpoint

     LD   420
     ST   State
     JMP state_machine_end
    no_setp_copy4:

  no_return_pause:

 STATE400_endif_A:
*///////////////////////////////////////////////////////////////////////////////
JMP state_machine_end
STATE400_end:

LD   State
EQ   410
JMPCN STATE410_end
STATE410:
*/////////////////////////////////////////////////////////////////////////////////
*// Wait Z reach the setpoint from inc movement
*/////////////////////////////////////////////////////////////////////////////////

 LD   xSurfSignalLock
 ANDN xSurfaceBusy
 JMPCN STATE410_endif_A

  LD   1
  S    yIncSetPReached

  LD   400
  ST   State

 STATE410_endif_A:
*///////////////////////////////////////////////////////////////////////////////
JMP state_machine_end
STATE410_end:

LD   State
EQ   420
JMPCN STATE420_end
STATE420:
*/////////////////////////////////////////////////////////////////////////////////
*// Wait the position is reached after return from hold
*/////////////////////////////////////////////////////////////////////////////////

 LD   xSurfSignalLock
 ANDN xSurfaceBusy
 JMPCN STATE420_endif_A

  LD   1
  R    yWait

  LD   1
  R    yIncSetPReached

  LD   310
  ST   State

 STATE420_endif_A:
*///////////////////////////////////////////////////////////////////////////////
JMP state_machine_end
STATE420_end:

* Jump L3 Between Sides
LD   State
EQ   430
JMPCN STATE430_end
STATE430:
*/////////////////////////////////////////////////////////////////////////////////
*// Jump L3 Request: VRTC is in simulation state, and must wait that interpolation
*// finish. Basically works like L5 but there is oly the interpolation of the
*// set-point but parabolic movement is done by the interpolator.
*/////////////////////////////////////////////////////////////////////////////////
 LD  xStartEx
 JMPCN no_start_jump1

  LD   1
  ST   yComRunning

  LD   6
  ST   yVPBSelect

  LD   1
  S    y_S_SimEnab              * Surface vrtc in Simulation

* Calculate vector A

  LD   xActual_X_Posit
  SUB  xInit_X_Posit                 * X init jump position
  DIV  100
  ABS
  ST   ActualXDist_A

  LD   xActual_Y_Posit
  SUB  xInit_Y_Posit                 * Y init jump position
  DIV  100
  ABS
  ST   ActualYDist_A

  LD   xActual_Z_Posit
  SUB  xInit_Z_Posit                 * Z init jump position
  DIV  100
  ABS
  ST   ActualZDist_A

  LD   xActual_C_Posit
  SUB  xInit_C_Posit                 * C init jump position
  DIV  100
  ABS
  ST   ActualCDist_A

* || A ||

  LD   ActualXDist_A
  MUL  ActualXDist_A
  ADD (
  LD   ActualYDist_A
  MUL  ActualYDist_A
  )
  ADD (
  LD   ActualZDist_A
  MUL  ActualZDist_A
  )
  ADD (
  LD   ActualCDist_A
  MUL  ActualCDist_A
  )
  ST   Actual_Dist_A

  LD   Actual_Dist_A
  SQRT
  ST   Actual_Dist_A

* Calculate vector B

  LD   xActual_X_Posit
  SUB  xNextPos_X_Jump                 * X Next jump position
  DIV  100
  ABS
  ST   ActualXDist_B

  LD   xActual_Y_Posit
  SUB  xNextPos_Y_Jump                 * Y Next jump position
  DIV  100
  ABS
  ST   ActualYDist_B

  LD   xActual_Z_Posit
  SUB  xNextPos_Z_Jump                 * Z Next jump position
  DIV  100
  ABS
  ST   ActualZDist_B

  LD   xActual_C_Posit
  SUB  xNextPos_C_Jump                 * C Next jump position
  DIV  100
  ABS
  ST   ActualCDist_B

* || B ||

  LD   ActualXDist_B
  MUL  ActualXDist_B
  ADD (
  LD   ActualYDist_B
  MUL  ActualYDist_B
  )
  ADD (
  LD   ActualZDist_B
  MUL  ActualZDist_B
  )
  ADD (
  LD   ActualCDist_B
  MUL  ActualCDist_B
  )
  ST   Actual_Dist_B

  LD   Actual_Dist_B
  SQRT
  ST   Actual_Dist_B

* Par = (|| A ||) / ( || A || + || B || )

  LD   Actual_Dist_A
  MUL  100
  DIV  (
  LD   Actual_Dist_A
  ADD  Actual_Dist_B
  )
  ST   Par

  LD   xPrevSetp                      * setpoint before jump
  DIV  10
  ST   y_S_SetPoint
  ST   %M184

  LD   xNextSetp                * Setpoint after jump
  SUB  xPrevSetp                * setpoint before jump
  ST   DeltaSetPoint

  *LD   ActualDistTot
  *MULDIV (M=DeltaSetPoint,D=DistTot) ** total distance for jump
  *DIV  10                            *cmm
  *ST   ZLinInterp

  LD   Par
  MULDIV (M=DeltaSetPoint,D=100) ** total distance for jump
  DIV  10                            *cmm
  ST   ZLinInterp

  LD   xPrevSetp                * setpoint before jump
  DIV  10
  ADD  ZLinInterp
  ST   y_T_SetPoint

  LD   Par
  GE   100
  *ST   %M189.1
  ST   yL3SetpointReached

 no_start_jump1:

 LDN  xJumpL3Req
 JMPCN no_end_jump1

  LD  1
  R   y_S_SimEnab                 * Surface vrtc in Simulation

  LD  3
  ST  yVPBSelect

  LD   ToolFlt_Q_FILTERED_DEL
  MULDIV(M=xCosBevelAngle,D=1000)
  ST  y_S_SetPoint

  LD  440
  ST  State
 no_end_jump1:

 JMP state_machine_end
STATE430_endif_A:
*///////////////////////////////////////////////////////////////////////////////
JMP state_machine_end
STATE430_end:

LD   State
EQ   440
JMPCN STATE440_end
STATE440:
*/////////////////////////////////////////////////////////////////////////////////
*// Wait the position is reached after jump
*/////////////////////////////////////////////////////////////////////////////////

 LD  1
 R   y_S_SimEnab                 * Surface vrtc in Simulation

 LD   ToolFlt_Q_FILTERED_DEL
 MULDIV(M=xCosBevelAngle,D=1000)
 ST  y_S_SetPoint

 LD   xSurfSignalLock
 ANDN xSurfaceBusy
 ANDN xStartEx
 JMPCN STATE440_endif_A

    LD   0
    ST   yComRunning

    LD   xNextSetp                * Setpoint after jump
    DIV  10
    ST   LastCutDistance

 *  LD   1                        * Reset bit to enable always regulation after jump
 *  R    RegFrozen

    LD   310
    ST   State
 JMP state_machine_end
STATE440_endif_A:
*///////////////////////////////////////////////////////////////////////////////
JMP state_machine_end
STATE440_end:

state_machine_end:
IDLE_end:

LD   State
ST   yState
ST   %M182

LD   y_S_SetPoint
ST   %M180

LD   y_T_SetPoint
ST   %M192

LD   LastCutDistance
ST   %M190

LD   xSetpoint
ST   %M191

END_FUNCTION_BLOCK

(* ---- SupForce.plc ---- *)
#funcdec "DynMng.plc"
#funcdec "FBAux.plc"

*//============================================================================
*// Force Following Support to be Down from ISO management
*//============================================================================

FUNCTION_BLOCK     ISO_SUP_FORCE_DOWN

VAR_INPUT
xIsoForce:         BOOL;      * iso_LsronCutting
xHoldMovSuperv:    BOOL;      * yHoldMovSuperv
END_VAR

VAR
Sup_Up_NotAllow:   BOOL;
R_TRIG_DWNCMD:     R_TRIG;
END_VAR

VAR_OUTPUT
yForceDwn:         BOOL;
END_VAR

CAL    R_TRIG_DWNCMD(CLK=xHoldMovSuperv)
LD     xIsoForce
AND    R_TRIG_DWNCMD.Q
S      Sup_Up_NotAllow

LDN    xIsoForce
ORN    %cn0.rc8.0
JMPCN  CLRSTATE
LD     %PLCFLAGS.0
ST     Sup_Up_NotAllow
CLRSTATE:

LD     Sup_Up_NotAllow
AND    xIsoForce
AND    %cn0.rc8.0
ST     yForceDwn

END_FUNCTION_BLOCK

*//============================================================================
*// In case of slave axis gearing state of G4010,
*// %ra92 == %ra24
*// PLC pre-stop quota need to be added (Estimated without JERK calculation)
*// CAL CALQ_PRESSLV(xEn:=,xQta:=,xSpdNum:=)
*// 0.5G 50000 Jerk as bench mark
*//============================================================================

FUNCTION_BLOCK     CALQ_PRESSLV

VAR_INPUT
xEn:               BOOL;
xQta:              DWORD;      * %ra4 / ra92
xSpdNum:           DWORD;      * The spline table number
END_VAR

VAR
tem_dis:           DWORD;
QtaCalc:           POINTS_INT_CALC;
END_VAR

VAR_OUTPUT
Q:                 DWORD;
END_VAR

LD     xQta
ST     Q

* Pre simpling data 0.5g 50000 Jerk，when RA92 fails

* speed > 2.2m/min and xQta < 1mm

LD     %ra115
MULDIV(M=60,D=1000)
GT     2200
AND(
       LD   xQta
       SUB  %ra24
	   LT   1000
)
JMPCN _ACT_LINERA
       LD   %ra115
       MULDIV(M=60,D=1000)
       ABS
       ST   QtaCalc.xPercSpeed            * Speed percentual value

       LD   1
       ST   QtaCalc.xCutLineInd           * cut line index (initial value 1 to 10)

       LD   xSpdNum
       ST   QtaCalc.xCodTec               * Tecnology 0=duty 1=power 2=frequency

       CAL  QtaCalc

       LD   QtaCalc.yResult               * Result
	   ST   tem_dis

	   LD   tem_dis
	   LT   0
	   JMPCN _SAFTY
	        LD  0
			ST  tem_dis
	   _SAFTY:

	   LD   tem_dis
	   ADD  xQta
       ST   Q

	   LDN  %ra3.2                        * Forward Movement of Slave Spindle
       ANDN %ra3.0
       JMPCN BCKWARDX1CASE
	        LD   xQta
            SUB  tem_dis
            ST   Q
       BCKWARDX1CASE:
_ACT_LINERA:

* Vel   Dis
* 2500	3020
* 5000	6320
* 7500	9965
* 10000	13955
* 12500	18297
* 15000	22985
* 17500	28020
* 20000	33400
* 22500	39128
* 25000	45200
* 27500	51626
* 30000	58396
* 32500	65516
* 35000	72980
* 37500	80792
* 40000	88950
* 42500	97459
* 45000	106313
* 47500	115513
* 50000	125000

PATH   %pd_splines[xSpdNum]

LD     %PLCFLAGS.8
JMPCN  _INIGLB
       LD  2
       ST  %pdh_interpType
       LD  21
       ST  %pdh_nPoints

       LD  0
       ST  %pdh_X0
       ST  %pdh_Y0

       LD  2500
       ST  %pdh_X1
	   LD  3020
       ST  %pdh_Y1

	   LD  5000
       ST  %pdh_X2
	   LD  6320
       ST  %pdh_Y2

	   LD  7500
       ST  %pdh_X3
	   LD  9965
       ST  %pdh_Y3

	   LD  10000
       ST  %pdh_X4
	   LD  13955
       ST  %pdh_Y4

	   LD  12500
       ST  %pdh_X5
	   LD  18297
       ST  %pdh_Y5

	   LD  15000
       ST  %pdh_X6
	   LD  22985
       ST  %pdh_Y6

	   LD  17500
       ST  %pdh_X7
	   LD  28020
       ST  %pdh_Y7

	   LD  20000
       ST  %pdh_X8
	   LD  33400
       ST  %pdh_Y8

	   LD  22500
       ST  %pdh_X9
	   LD  39128
       ST  %pdh_Y9

	   LD  25000
       ST  %pdh_X10
	   LD  45200
       ST  %pdh_Y10

	   LD  27500
       ST  %pdh_X11
	   LD  51626
       ST  %pdh_Y11

	   LD  30000
       ST  %pdh_X12
	   LD  58396
       ST  %pdh_Y12

	   LD  32500
       ST  %pdh_X13
	   LD  65516
       ST  %pdh_Y13

	   LD  35000
       ST  %pdh_X14
	   LD  72980
       ST  %pdh_Y14

	   LD  37500
       ST  %pdh_X15
	   LD  80792
       ST  %pdh_Y15

	   LD  40000
       ST  %pdh_X16
	   LD  88950
       ST  %pdh_Y16

	   LD  42500
       ST  %pdh_X17
	   LD  97459
       ST  %pdh_Y17

	   LD  45000
       ST  %pdh_X18
	   LD  106313
       ST  %pdh_Y18

	   LD  47500
       ST  %pdh_X19
	   LD  115513
       ST  %pdh_Y19

	   LD  50000
       ST  %pdh_X20
	   LD  125000
       ST  %pdh_Y20

_INIGLB:

END_FUNCTION_BLOCK

*//============================================================================
*// Cylinder Composite Support Calculation Based On Current Profile Shape
*// CAL CALC_CYCOMSUP(xLenCy:=, xEnCyTubeSiz:=)
*//============================================================================

FUNCTION_BLOCK     CALC_CYCOMSUP

VAR_INPUT
xLenCy:            DWORD;     * The stroke of cylinder [mm]
xEnCyTubeSiz:      DWORD;     * > Qta to disable cylinder [mm] (not the trave of servo because which could be different)
xAxNum:            DWORD;     * The servo support axis number
END_VAR

VAR
OutofRng:          BOOL;
X:                 DWORD;
Y:                 DWORD;
Radius:            DWORD;
inner:             DWORD;
outter:            DWORD;
temLenCy:          DWORD;
temAxtra:          DWORD;
CyTubeSiz:         DWORD;
MaxMin:          COMPARE;
END_VAR

VAR_OUTPUT
* Bit 0: Only Motor, offset == 0
* Bit 1: Both Cylinder and Motor, offset == Cylinder Stroke
* Bit 2: Impossible to always follow, msgout (Out of range, should not happen. Otherwise, tube is too large)
yModeCode:         DWORD;
END_VAR

LD     xLenCy
MUL    1000
ST     temLenCy

LD     xEnCyTubeSiz
MUL    1000
ST     CyTubeSiz

LD     %gIso23
MUL    1000
ST     X

LD     %gIso24
MUL    1000
ST     Y

CAL    MaxMin(A:=X,B:=Y)
LD     MaxMin.yMin
DIV    2
ST     inner

LD     0
HYPOT (X=X,Y=Y)
DIV    2
ST     outter

LD     %gIso25       *RAIDIUS UNIT DIFFERENT
ST     Radius

LD     %gIso26
EQ     0
JMPCN  _RECT
       LD  X
	   SUB Radius
	   ST  X

	   LD  Y
	   SUB Radius
	   ST  Y

       LD  0
       HYPOT(X=X,Y=Y)
	   DIV 2
       ADD Radius
	   ST  outter
_RECT:

LD     %gIso26
EQ     1
JMPCN  _ROUND
       LD  inner
	   ST  outter
_ROUND:

* Output

LD     0
ST     yModeCode

PATH   %ax[xAxNum]

LD     %pa22
SUB    %pa21
ST     temAxtra

LD     outter
SUB    inner
GT(
LD     temAxtra
SUB    temLenCy
)
AND(
LD     temLenCy
GT     inner
)
AND(
LD     temLenCy
LT     outter
)
ST     OutofRng

LD     outter
GT     CyTubeSiz
ST     yModeCode.0
STN    yModeCode.1

LD     OutofRng
ST     yModeCode.2

END_FUNCTION_BLOCK

(* ---- suppFB.plc ---- *)
*******************************************************************************
*   suppFB.plc
*   ESAutomotion
*   LASER machine
*******************************************************************************
#funcdec "assi.plc"

*******************************************************************************
*   Support axis management (Cascading Blend Switch, G.D)
*******************************************************************************

VAR_IN_OUT
AxPos             AT  %ra4;      * Axis position
Go_Follow         AT  %rgau0;    * Force down by blending algh.
AddFollow         AT  %rgau1;    * Add value during following
BldState          AT  %rgau2;    * Blend switch output, (0->1000) (parking -> following)
ParkingSet        AT  %rgau3;    * Real time parking position (input)
AddFollow_Out     AT  %rgau4;    * Add value during following (output)
ParkingSet_Out    AT  %rgau5;    * Real time parking position (output)

filterT1Rate      AT  %rgdau0;   * Blendswitch filter rate [0.001/min]
addValueVel       AT  %rgdau1;   * Following add value speed [um/min]
addValueVelM      AT  %rgdau2;   * Parking speed [um/min]

ProbeThreshold    AT  %gIso30;   *(gIso30) probe threshold (G2292)

LatCenterToCloseRun AT %SUPPORTS_SYSTEM.values13.17;
END_VAR

FUNCTION_BLOCK    SUPPORT

VAR_INPUT
xUaxDir:          BOOL;          * 1 - if spindle move towards the 0 of the machine decreasing its quota
                                 * 0 - if spindle move towards the 0 of the machine increasing its quota
xHoldExem:        BOOL;          * Support Hold Exemption (in case of initialization)
xUaxStill:        BOOL;          * U axis is not moving (%ra3.0)
xReset:           BOOL;          * Emergency and Reset for PosAx
xEnabAutoDwn:     BOOL;          * Enable Auto Support Down
xEnabAutoUp:      BOOL;          * Enable Auto Support Up (Blend)
xBlendSwitchEn:   BOOL;          * blendswitch enable
xParkCmd:         BOOL;          * JOG / Auto Cmd to park
xSensSafePos:     BOOL;          * Safety sensor to be sure the support is parked
xEnSecFollow:     BOOL;          * Enable addvalue during support following
xG520VSup:        BOOL;          * In G520 using V support unloading (Parking Target by ISO)
xEnCyComSup:      BOOL;          * Enable motor cylinder composite support
xEnBldFeed:       BOOL;          * Blend switch feedrate management

xSupervisePos:   DWORD;          * Position of the U axis -> start autodown
xSuperviseOft:   DWORD;          * Offset of position U to be closer to the support
xLimitSuppDwn:   DWORD;          * U axis limit position for support down
xParkingPos:     DWORD;          * Support Parking position
xUnSupQta:       DWORD;          * Support Parking position to Unload
xAddFollPos:     DWORD;          * Added following targets
xCyComOft:       DWORD;          * Motor cylinder composite support blend switch offset
xM700_M704:      DWORD;          * M700, M704 executing
xBlendId:        DWORD;          * Blend ID for speed reset ([lv, lat, ulv, uhor]=[0,1,2,3])
xBldFeed:        DWORD;          * Blend switch feedrate % (0-100)
END_VAR

VAR_OUTPUT
yReqGrant:        BOOL;
yHoldMovSupp:     BOOL;
yHoldMovSuperv:   BOOL;
yAxInParkPos:     BOOL;
yCenterOpen:      BOOL;
yCyComDwn:        BOOL;
yCyComOft:       DWORD;
END_VAR

VAR
resReq:           BOOL;
Req_Parking:      BOOL;
HoldSuppAxis:     BOOL;
HoldSuperviAxis:  BOOL;
appoggio:         BOOL;
GoUpSuppAuto:     BOOL;
M700Running:      BOOL;
M704Running:      BOOL;
CenterOpen:       BOOL;

OuterPlusOne:     DWORD;
Supervise_Oft:    DWORD;
ProbeThrsTmp:     DWORD;

TON_CLOSE_LOOP:    TON;
TRIG_PRKCON:      TRIG;
R_TRIG_BLD:     R_TRIG;
R_RES_REQ:      R_TRIG;
RTRIG_REQ_PARK: R_TRIG;
RTRIG_PARK:     R_TRIG;
RTRIG_RES_PARK: R_TRIG;
RTRIG_SAFE_DWN: R_TRIG;
RTRIG_REQ_UP:   R_TRIG;
RTRIG_RES_UP:   R_TRIG;
FTRIG_PRGRUN:   F_TRIG;
PosSupp:      AX_POSIZ;
END_VAR

LD   xM700_M704
EQ   700
AND  %cn0.rc8.0
ST   M700Running

LD   xM700_M704
EQ   704
AND  %cn0.rc8.0
ST   M704Running

LD   ProbeThreshold
ST   ProbeThrsTmp

* Motor cylinder composite support type
LD   xEnCyComSup
JMPCN _CYCOMEN
     LD   xCyComOft
     ADD  ProbeThreshold
     ST   ProbeThrsTmp
_CYCOMEN:

* ProbeThreshold = Optimized_lift = OuterPlusOne + 20
LD   ProbeThrsTmp
SUB  19000           *19mm
ST   OuterPlusOne

LDN  xEnSecFollow
JMPCN CLRFOFFSET
     LD   0
	 ST   AddFollow
CLRFOFFSET:

* Added offset within safely down distance
LD   xSuperviseOft
ABS
ST   Supervise_Oft

LD   xSuperviseOft
ABS
GT   200000
JMPCN OUTRNGOFT
     LD   xSuperviseOft
	 ABS
     ST   Supervise_Oft
OUTRNGOFT:

CAL  TON_CLOSE_LOOP (IN:=%ra0.0,PT:=300)

LDN  xUaxDir
JMPCN  no_check
     * Supervisor
     LD   xSupervisePos
     GT   xLimitSuppDwn
     AND  TON_CLOSE_LOOP.Q
     ANDN (
     LD   AxPos
     ADD  1000
     GT   xParkingPos
     *AND  xSensSafePos
     )
     ST   HoldSuperviAxis

     LD   xSupervisePos
     ADD  200000                       * safety
	 SUB  Supervise_Oft
     GT   xLimitSuppDwn
     AND  TON_CLOSE_LOOP.Q
     ANDN HoldSuperviAxis
     ST   HoldSuppAxis

	 LD   xSupervisePos
	 ADD  350000
	 GT   xLimitSuppDwn
	 ANDN (
     LD   AxPos
     ADD  1000
     GT   xParkingPos
     )
	 ANDN xUaxStill
	 OR(
	 LDN  %ra3.0
	 ANDN LatCenterToCloseRun
	 )
	 ST   CenterOpen
no_check:

LD   xUaxDir
JMPCN  no_check1
     * Supervisor
     LD   xSupervisePos
     LT   xLimitSuppDwn
     AND  TON_CLOSE_LOOP.Q
     ANDN (
     LD   AxPos
     ADD  1000
     GT   xParkingPos
     *AND  xSensSafePos
     )
     ST   HoldSuperviAxis

     LD   xSupervisePos
     SUB  200000                       * safety
	 ADD  Supervise_Oft
     LT   xLimitSuppDwn
     AND  TON_CLOSE_LOOP.Q
     ANDN HoldSuperviAxis
     ST   HoldSuppAxis

	 LD   xSupervisePos
	 SUB  350000
	 LT   xLimitSuppDwn
	 ANDN (
     LD   AxPos
     ADD  1000
     GT   xParkingPos
     )
	 ANDN xUaxStill
	 OR(
	 LDN  %ra3.0
	 ANDN LatCenterToCloseRun
	 )
	 ST   CenterOpen
no_check1:

LD   HoldSuppAxis
OR(
     LD   HoldSuperviAxis
     ANDN HoldSuppAxis
)
ANDN %cn0.rc8.0
ST   appoggio
CAL  RTRIG_SAFE_DWN(CLK:=appoggio)

CAL  RTRIG_REQ_PARK (CLK:=HoldSuppAxis)
CAL  RTRIG_PARK (CLK:=xParkCmd)
LD   RTRIG_REQ_PARK.Q
OR   RTRIG_SAFE_DWN.Q
AND  xEnabAutoDwn
OR   RTRIG_PARK.Q
ANDN %rc0.8                 *in ref
AND  TON_CLOSE_LOOP.Q
S    Req_Parking

*//============================================================================
*// JOG Mode Supports Parking
*//============================================================================
LDN   %cn0.rc8.0
OR(
LD    xParkCmd
OR    Req_Parking
ANDN  xBlendSwitchEn
AND   %cn0.rc8.0
)
JMPCN Jog_management
      LD   Req_Parking
      AND  TON_CLOSE_LOOP.Q
      ANDN PosSupp.yax_ENDERR
      ST   PosSupp.xax_ENABLE
	  CAL  TRIG_PRKCON(CLK=PosSupp.xax_ENABLE)

      LDN  PosSupp.xax_ENABLE
	  OR   TRIG_PRKCON.Q
      ST   PosSupp.xax_CLEAR

      LD   PosSupp.xax_ENABLE
      AND  PosSupp.yax_READY
      ANDN PosSupp.yax_ENDERR
      ST   PosSupp.xax_START

      LD   xParkingPos
      ST   PosSupp.xax_QUOTA

      LD   %pa9
      ST   PosSupp.xax_VEL

      CAL  PosSupp

      LD   PosSupp.yax_ENDOK
      OR   xReset
      ST   resReq

      CAL  R_RES_REQ (CLK:=resReq)
      LD   R_RES_REQ.Q
      R    Req_Parking
Jog_management:

CAL   FTRIG_PRGRUN (CLK:=%cn0.rc8.0)
LD    FTRIG_PRGRUN.Q
R     Req_Parking

*//============================================================================
*// Blendswitch Veladdval / Hold / Feedrate Condition initialization
*//============================================================================
LD   %BLEND_VEL.filTRate[xBlendId]
ST   filterT1Rate

LD   %BLEND_VEL.velAddVal[xBlendId]
ST   addValueVel
ST   addValueVelM

LD   xEnBldFeed
JMPCN _BLENDFEED
	  LD   xBldFeed
	  MULDIV(M=filterT1Rate,D=100)
	  ST   filterT1Rate

	  LD   xBldFeed
	  MULDIV(M=addValueVel,D=100)
	  ST   addValueVel
      ST   addValueVelM
_BLENDFEED:

LD    %cn0.rc8.1
AND   xBlendSwitchEn
JMPCN _BLENDHOLD
      LD   0
      ST   filterT1Rate
      ST   addValueVel
      ST   addValueVelM
_BLENDHOLD:

*//============================================================================
*// Auto Mode Supports (Bi-State CMD)
*//============================================================================
LD    %cn0.rc8.0
AND   xBlendSwitchEn
AND   xEnabAutoDwn
JMPCN AUTO_MANAGEMENT
      LD   HoldSuppAxis
	  OR(
	       LD   HoldSuperviAxis
           ANDN HoldSuppAxis
	  )
      OR   xParkCmd
	  OR   Req_Parking
      JMPCN BLEND_PARK_STATUS             *++++++
           LD   0
           ST   Go_Follow
		   LD   0
		   ST   AddFollow

		   * Cascading Movement after bld = 0
		   LD   BldState
		   EQ   0
		   ANDN M700Running
		   ANDN M704Running
		   ANDN xG520VSup
		   JMPCN PARKLVL0
		         LD   xParkingPos
		         ST   ParkingSet
		   PARKLVL0:

		   * V support leveling in G520 -> xG520VSup
		   * At the moment, ParkingSet given by ISO only
		   LD   BldState
		   EQ   0
		   ANDN M700Running
		   ANDN M704Running
		   AND  xG520VSup
		   JMPCN PARKUNLOAD
		         LD   xUnSupQta
		         ST   ParkingSet
		   PARKUNLOAD:

		   * During G0 and M700
		   LD   BldState
		   EQ   0
		   AND  M700Running
		   AND (
				LD   OuterPlusOne
				ADD  200                 *0.2mm
				GT   AxPos
		   )
           ANDN (
		   		LD   HoldSuperviAxis
                ANDN HoldSuppAxis
		   )
		   JMPCN PARKLVL1
		        LD   ProbeThrsTmp
		        ST   ParkingSet
		   PARKLVL1:

		   * In case of X moves causes hold in M700
		   LD   HoldSuperviAxis
           ANDN HoldSuppAxis
		   AND  M700Running
		   JMPCN OPTPRKHOLD
				 LD   xParkingPos
		         ST   ParkingSet
		   OPTPRKHOLD:

      JMP  BLEND_SKIP_FOLLOW              *//////
      BLEND_PARK_STATUS:                  *++++++

	       LD   xEnabAutoUp
		   JMPCN STATUS_ENUP
		         LD   OuterPlusOne
		         ST   ParkingSet

                 LD   1
				 AND(
				 LD   ParkingSet
				 EQ   ParkingSet_Out
				 )
                 ST   Go_Follow
		   STATUS_ENUP:

		   * Added value management following
		   LD    BldState
		   EQ    1000
		   AND   xEnSecFollow
		   JMPCN STATUS_FOFFSET
		         LD   xAddFollPos
			     ST   AddFollow
		   STATUS_FOFFSET:

      BLEND_SKIP_FOLLOW:                  *//////

      LD   %PLCFLAGS.0
      ST   Req_Parking
AUTO_MANAGEMENT:

LDN   %cn0.rc8.0
JMPCN RSTBLEND
      LD    0
      ST    Go_Follow
RSTBLEND:

*//============================================================================
*// Output
*//============================================================================
LD    AxPos
SUB   xParkingPos
ABS
LT    1000
ST    yAxInParkPos

LD    Req_Parking
ANDN  %cn0.rc8.0
OR(
LD    xParkCmd
OR    Req_Parking
ANDN  xBlendSwitchEn
AND   %cn0.rc8.0
)
AND   TON_CLOSE_LOOP.Q
ANDN (
LD    xHoldExem
ANDN  xBlendSwitchEn
AND   %cn0.rc8.0
)
ST    yReqGrant

LD    HoldSuppAxis
ANDN (
LD    xHoldExem
ANDN  xBlendSwitchEn
AND   %cn0.rc8.0
)
ANDN  yReqGrant
OR(
LD    %cn0.rc9                * Registro funzioni M canale 0
EQ    30
AND   %cn0.rc8.4              * Strobe funzioni M canale 0
)
ST    yHoldMovSupp

LD    HoldSuperviAxis
ST    yHoldMovSuperv

LD    CenterOpen
OR(
LD    xM700_M704
NE    0
)
ST    yCenterOpen

LD    xCyComOft
EQ    0
AND   xEnCyComSup
ST    yCyComDwn

LD    0
ST    yCyComOft

LD   xEnCyComSup
JMPCN _CYCOMENOFT
     LD   xCyComOft
     ST   yCyComOft
_CYCOMENOFT:

END_FUNCTION_BLOCK

(* ---- WorkList.plc ---- *)
*******************************************************************************
*   WORKLIST.PLC
*   ESAutomotion
*   LASER machine
*******************************************************************************
#funcdec "assi.plc"
#funcdec "mand.plc"
#funcdec "cnc.plc"

VAR
#include "assi.inc"
#include "cnc.inc"
END_VAR

#include "iol.inc"

VAR_IN_OUT

#include "mem.inc"

TIMER_PROG          AT %wl_time;                    * timer
SEQ_VIS             AT %WlistMngt.wl_mngdwpar0;     * (WlistMngt.wl_mngdwpar0)Sequenza per vis.
CMD_CHCOMP          AT %CompData0;                  * Comando canale computazionale
WENDL               AT %wl_endl;
WPARA               AT %wl_parA0;
END_VAR

*******************************************************************************
*   FB GESTIONE LISTE
*   (#WLIST)
*******************************************************************************
FUNCTION_BLOCK WORK_LIST

VAR_INPUT
xEnable:            BOOL;           ** abilitazione
xProgRun:           BOOL;           ** program run
xEmissionOn:        BOOL;           ** Laser acceso (O_O_A2_LASER_PROG_RUN)
END_VAR

VAR_OUTPUT
END_VAR

VAR
F_TRIGP:            F_TRIG;     * Program run down
L_RTRIG_NEXT:       R_TRIG;     * Vis. prog successivo
L_RTRIG_PREV:       R_TRIG;     * Vis. prog precedente
L_RTRIG_1SEC:       R_TRIG;     * Cadenza di 1 secondo
RefreshGraph:       BOOL;
L_appoggio:         BOOL;       * appoggio
L_PrevUiplPage:     DWORD;      * Pagina precedente UIPL
CopyVal_SEQ_VIS:    DWORD;      * Copia numero sequenza vis.
END_VAR
*******************************************************************************

***************************************
* List running
***************************************
LD   0
ST   %WlistMngt.wl_ListRunning

LD   xEnable
AND  xProgRun
JMPCN No_Run

LD   1
ST   %WlistMngt.wl_ListRunning

No_Run:

***************************************
* Gestione visualizzazione linea
***************************************
LD   %Uipl.Field
EQ   9999
ANDN %WlistMngt.wl_ListRunning
ANDN GRAPH_DRAW_RUN                ** ui33.7 Graphics drawing in progress
AND (
LD   SEQ_VIS                       ** (WlistMngt.wl_mngdwpar0)Sequenza per vis.
NE   %Uipl.Row
)
JMPCN NoSel

LD   %Uipl.Row
ST   SEQ_VIS                       ** (WlistMngt.wl_mngdwpar0)Sequenza per vis.

NoSel:
***************************************
* Rinfresco grafica
***************************************
LD   ALWAYS_ZERO                   ** PLCFLAGS.0  Flag sempre stato off
ST   RefreshGraph

LD   SEQ_VIS                       ** (WlistMngt.wl_mngdwpar0)Sequenza per vis.
EQ   CopyVal_SEQ_VIS               ** Copia numero sequenza vis.
JMPC AGGNUMCODE

LD   SEQ_VIS                       ** (WlistMngt.wl_mngdwpar0)Sequenza per vis.
ST   CopyVal_SEQ_VIS               ** Copia numero sequenza vis.

LD   ALWAYS_ONE                    ** PLCFLAGS.1  Flag sempre stato on
ST   RefreshGraph

AGGNUMCODE:
LD   L_PrevUiplPage                ** Pagina precedente UIPL
EQ   5000                   ** Numero pagina della LISTA lavoro
AND (
LD   %Uipl.Page
NE   5000                   ** Numero pagina della LISTA lavoro
)
OR (
LD   L_PrevUiplPage                ** Pagina precedente UIPL
EQ   5001                   ** Numero pagina GRAFICA FULL SCREEN
AND (
LD   %Uipl.Page
NE   5001                   ** Numero pagina della LISTA lavoro
)
)
ST   L_appoggio                    ** appoggio

LD   %Uipl.Page
ST   L_PrevUiplPage                ** Pagina precedente UIPL

CAL  F_TRIGP(CLK=PRGRUN_CN0)       ** Program run down

LD   L_appoggio                    ** appoggio
OR   %SoftBtn0.0                   ** Reset PIECE and GEOMETRY
OR   RefreshGraph
OR   ON_ONE_SCAN                   ** PLCFLAGS.8  Flag on alla prima scansione PLC
OR   Pul_Reset                     ** (gPlc0.3)Reset pushbutton
OR   F_TRIGP.Q
AND  %LSRPlcOp0.5                  ** Worklist mode enabled
JMPCN NoSendCmd

LD   5                          * Comando refresh grafica (canale computazionale)
ST   CMD_CHCOMP                    ** Comando canale computazionale

NoSendCmd:
***************************************
* Lock editing in pagina EDITOR LISTE
***************************************
LD   %WlistMngt.wl_ListRunning
ST   %WlistMngt.wl_EditLock

***************************************
* Gestione TEMPI di esecuzione
***************************************
CAL L_RTRIG_1SEC(CLK=NORMAL_BLINK) ** Cadenza di 1 secondo

PATH %Wlist[%WlistMngt.wl_Index]

LD   %cn0.rc8.0                    * Programma in corso cn0
ANDN PRGSTOP_CN0                   ** (cn0.rc8.1)  Programma interrotto CN0
**AND  xEmissionOn  *todomag scommentare nel caso serva il tempo sull'accensione laser
AND  L_RTRIG_1SEC.Q
AND (
LD   %WlistMngt.wl_ListRunning
EQ   1
)
JMPCN NoIncTimer

LD   TIMER_PROG                    ** timer
ADD  1
ST   TIMER_PROG                    ** timer

NoIncTimer:

END_FUNCTION_BLOCK
